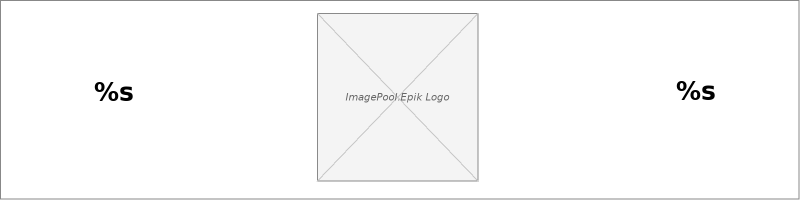
VISUALIZATION Header  // 800x200
    Image (317,13 161x168), image: ImagePool.Epik Logo
    Textfield (601,41 190x99), "%s", text variable: GVL.SystemTime
    Textfield (8,43 212x97), "%s", text variable: GVL.SystemDate
END_VISUALIZATION

(* stored: Version 1.1.0.1, ProductVersion 3.1.4024.12
   Visu Header: Id {3c45c616-a311-49f3-b412-6c37ee47343b} *)
